{attribute 'linkalways'} 
{attribute 'no_explicit_call' := 'This FB is a CLASS and must be accessed using methods or properties'}
{attribute 'enable_dynamic_creation'}
FUNCTION_BLOCK QueueDisposedEvent EXTENDS QueueEvent IMPLEMENTS I_QueueDisposedEvent

END_FUNCTION_BLOCK

(* stored: Version 1.1.0.1, ProductVersion 3.1.4024.12
   POU QueueDisposedEvent: Id {1d08acbe-a9bc-4776-a7fc-05c3459acae3}, SpecialFunc None *)
